# EPICS substitutions: test/simulatorApp/Db/sim_4096.substitutions
file "sim_0256.db" {
pattern { R }
{ "\$(R)0" }
{ "\$(R)1" }
{ "\$(R)2" }
{ "\$(R)3" }
{ "\$(R)4" }
{ "\$(R)5" }
{ "\$(R)6" }
{ "\$(R)7" }
{ "\$(R)8" }
{ "\$(R)9" }
{ "\$(R)A" }
{ "\$(R)B" }
{ "\$(R)C" }
{ "\$(R)D" }
{ "\$(R)E" }
{ "\$(R)F" }
}
